FUNCTION_BLOCK FB_TCMotor
VAR_INPUT
END_VAR
VAR_OUTPUT
END_VAR
VAR
	fb_TC_Ap							: DFB_Cylinder;
	_Col_PCWValve_Perm					: WORD;
	_Col_PCWValve_SD									: WORD;
	
	_DUT_TC_e						: DUT_Cylinder;
END_VAR

ACTION PermSD:

END_ACTION

END_FUNCTION_BLOCK

(* stored: Version 1.1.0.1, ProductVersion 3.1.4022.18
   POU FB_TCMotor: Id {541e675d-c901-46ef-8343-e944626c84c3}, SpecialFunc None
   Action PermSD: Id {5e1c502e-582d-4762-86b5-bbeb6cc40854} *)
